TYPE ST_ManipAxis :
STRUCT

(* Controls *)
xEnable	:	BOOL := TRUE;
rReqAbsPos	:	REAL;
rReqRelPos	:	REAL;
xStart	:	BOOL;
xStop	:	BOOL;
wMode	:	E_AxisMoveMode;
//EPICS motor status
uiMsta	:	UINT;
//EPICS Position readback
rActPos	:	REAL;
//Axis enabled readback
xEnabled	:	BOOL;
	
(* Axis motor *)
stAxis	:	AXIS_REF;
lrVelocity	:	LREAL	:=1; //mm/s

eState	:	E_AxisMotionState;

xHiLS	AT %I* :	BOOL;
xLoLS	AT %I* :	BOOL;

END_STRUCT
END_TYPE

(* stored: Version 1.1.0.1, ProductVersion 3.1.4020.12
   DUT ST_ManipAxis: Id {8a2b69b2-0749-42c2-bd32-ad09794455d6} *)
